Universal Robots PolyScope program: 28-pickAndPlace.urp

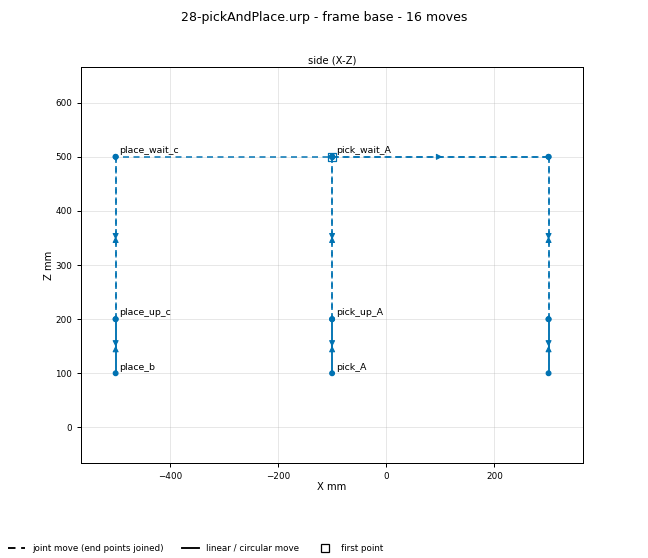
[picture p0: tool path of 28-pickAndPlace.urp in frame base, 16 of 16 moves have a stored position in this frame; points joined in program order, loops and branches not executed]
ProgramRoot directory=/home/ur/ursim-3.1/programs/basic training/28-pickAndPlace; kinematics=(a=[0, -0.425, -0.39225, 0, 0, 0], d=[0.08916, 0, 0, 0.10915, 0.09465, 0.0823], alpha=[1.5708, 0, 0, 1.5708, -1.5708, 0], deltaTheta=[0, 0, 0, 0, 0, 0], status=notInitialized); lastSavedInVersion=(project__name=Polyscope, major__version=3, minor__version=1, svn__revision=17195, build__date=Mar 11 2015, 13:02:28); name=28-pickAndPlace; programVersion=(project__name=Polyscope, major__version=3, minor__version=1, svn__revision=17195, build__date=Mar 11 2015, 13:02:28); robotEnvironmentFileName=default; serialNumberRobot=2014350001
  BeforeStart description=COMMAND_SEQUENCE_BEFORE_PROGRAM_START; name=BeforeStart
    Move cartesianAcceleration=1.2; cartesianSpeed=0.25; jointAcceleration=1.3962634015954636; jointSpeed=1.0471975511965976; sharedProcessMoveBlendRadius=0.025; motionType=JOINT_SPACE
      Waypoint blendRadius=0.05; cartesianAcceleration=1.2; cartesianSpeed=0.25; jointAcceleration=1.3962634015954636; jointSpeed=1.0471975511965976; nextMotionTime=2.0; stoppoint=true; useSharedBlendParameter=true; useSharedParameters=true; outputFlangePose=(pos=(x=-0.09999996819589972, y=-0.4000000526540407, z=0.5000000010103537), rot=(x=-0.0012210995530382433, y=3.1162764787073605, z=0.038892320957760594)); position=TCP in base x=-100 y=-400 z=500 mm, rx=-0.0012 ry=3.1163 rz=0.0389 rad; joints [-88.988, -79.302, -89.258, -102.845, 91.461, 0.95] deg; positionType=FIXED_POSITION; waypointPoseInFeatureCoordinates=(pos=(x=-0.0999999669318244, y=-0.4000001276702773, z=0.499999972698533), rot=(x=-0.0012210995530382489, y=3.1162764787073782, z=0.0388923209577583)); name=pick_wait_A
  MainProgram cartesianAcceleration=1.2; cartesianSpeed=0.25; jointAcceleration=1.3962634015954636; jointSpeed=1.0471975511965976; sharedProcessMoveBlendRadius=0.025; motionType=JOINT_SPACE
    If expr=ExpressionIONode; type=IF_NODE
      CallSubProgram subProgramNodeToCall=(SubProgramNode=(default=(keepHidden=false, keepSynchrnized=false, trackProgramExecution=false, name=sub_b)))
    If type=ELSE_NODE
      CallSubProgram subProgramNodeToCall=(SubProgramNode=(default=(keepHidden=false, keepSynchrnized=false, trackProgramExecution=false, name=sub_c)))
    CallSubProgram subProgramNodeToCall=(SubProgramNode=(default=(keepHidden=false, keepSynchrnized=false, trackProgramExecution=false, name=sub_a)))
  Event expression=ExpressionIONode
    Wait 
    Set 
  SubProgram name=sub_a
    Move cartesianAcceleration=1.2; cartesianSpeed=0.25; jointAcceleration=1.3962634015954636; jointSpeed=1.0471975511965976; sharedProcessMoveBlendRadius=0.025; motionType=JOINT_SPACE
      Waypoint blendRadius=0.05; cartesianAcceleration=1.2; cartesianSpeed=0.25; jointAcceleration=1.3962634015954636; jointSpeed=1.0471975511965976; nextMotionTime=2.0; stoppoint=true; useSharedBlendParameter=true; useSharedParameters=true; outputFlangePose=(pos=(x=-0.09999996819589972, y=-0.4000000526540407, z=0.5000000010103537), rot=(x=-0.0012210995530382433, y=3.1162764787073605, z=0.038892320957760594)); position=TCP in base x=-100 y=-400 z=500 mm, rx=-0.0012 ry=3.1163 rz=0.0389 rad; joints [-88.988, -79.302, -89.258, -102.845, 91.461, 0.95] deg; positionType=FIXED_POSITION; waypointPoseInFeatureCoordinates=(pos=(x=-0.0999999669318244, y=-0.4000001276702773, z=0.499999972698533), rot=(x=-0.0012210995530382489, y=3.1162764787073782, z=0.0388923209577583)); name=pick_wait_A
      Waypoint blendRadius=0.05; cartesianAcceleration=1.2; cartesianSpeed=0.25; jointAcceleration=1.3962634015954636; jointSpeed=1.0471975511965976; nextMotionTime=2.0; stoppoint=true; useSharedBlendParameter=true; useSharedParameters=true; outputFlangePose=(pos=(x=-0.09999996693182436, y=-0.40000012767028115, z=0.2000000005382103), rot=(x=-0.0012210995530365215, y=3.116276478707369, z=0.03889232095774556)); position=TCP in base x=-100 y=-400 z=200 mm, rx=-0.0012 ry=3.1163 rz=0.0389 rad; joints [-88.988, -88.3, -127.491, -55.614, 91.461, 0.95] deg; positionType=FIXED_POSITION; waypointPoseInFeatureCoordinates=(pos=(x=-0.09999996819589951, y=-0.40000005265404437, z=0.1999999632555712), rot=(x=-0.0012210995530369398, y=3.1162764787073427, z=0.0388923209577584)); name=pick_up_A
    Move cartesianAcceleration=1.2; cartesianSpeed=0.25; jointAcceleration=1.3962634015954636; jointSpeed=1.0471975511965976; sharedProcessMoveBlendRadius=0.025; motionType=CARTESIAN_SPACE
      Waypoint blendRadius=0.05; cartesianAcceleration=1.2; cartesianSpeed=0.25; jointAcceleration=1.3962634015954636; jointSpeed=1.0471975511965976; nextMotionTime=2.0; stoppoint=true; useSharedBlendParameter=true; useSharedParameters=true; outputFlangePose=(pos=(x=-0.0999999681958997, y=-0.4000000526540418, z=0.10000000081214921), rot=(x=-0.0012210995530447125, y=3.1162764787073605, z=0.038892320957759144)); position=TCP in base x=-100 y=-400 z=100 mm, rx=-0.0012 ry=3.1163 rz=0.0389 rad; joints [-88.988, -101.017, -134.096, -36.292, 91.461, 0.95] deg; positionType=FIXED_POSITION; waypointPoseInFeatureCoordinates=(pos=(x=-0.09999996708411972, y=-0.40000011440850547, z=0.10000011559988649), rot=(x=-0.0012211090279065008, y=3.1162764797380107, z=0.03889157798959221)); name=pick_A
      Waypoint blendRadius=0.05; cartesianAcceleration=1.2; cartesianSpeed=0.25; jointAcceleration=1.3962634015954636; jointSpeed=1.0471975511965976; nextMotionTime=2.0; stoppoint=true; useSharedBlendParameter=true; useSharedParameters=true; outputFlangePose=(pos=(x=-0.09999996693182436, y=-0.40000012767028115, z=0.2000000005382103), rot=(x=-0.0012210995530365215, y=3.116276478707369, z=0.03889232095774556)); position=TCP in base x=-100 y=-400 z=200 mm, rx=-0.0012 ry=3.1163 rz=0.0389 rad; joints [-88.988, -88.3, -127.491, -55.614, 91.461, 0.95] deg; positionType=FIXED_POSITION; waypointPoseInFeatureCoordinates=(pos=(x=-0.09999996819589951, y=-0.40000005265404437, z=0.1999999632555712), rot=(x=-0.0012210995530369398, y=3.1162764787073427, z=0.0388923209577584)); name=pick_up_A
    Move cartesianAcceleration=1.2; cartesianSpeed=0.25; jointAcceleration=1.3962634015954636; jointSpeed=1.0471975511965976; sharedProcessMoveBlendRadius=0.025; motionType=JOINT_SPACE
      Waypoint blendRadius=0.05; cartesianAcceleration=1.2; cartesianSpeed=0.25; jointAcceleration=1.3962634015954636; jointSpeed=1.0471975511965976; nextMotionTime=2.0; useSharedParameters=true; outputFlangePose=(pos=(x=-0.09999996819589972, y=-0.4000000526540407, z=0.5000000010103537), rot=(x=-0.0012210995530382433, y=3.1162764787073605, z=0.038892320957760594)); position=TCP in base x=-100 y=-400 z=500 mm, rx=-0.0012 ry=3.1163 rz=0.0389 rad; joints [-88.988, -79.302, -89.258, -102.845, 91.461, 0.95] deg; positionType=FIXED_POSITION; waypointPoseInFeatureCoordinates=(pos=(x=-0.0999999669318244, y=-0.4000001276702773, z=0.499999972698533), rot=(x=-0.0012210995530382489, y=3.1162764787073782, z=0.0388923209577583)); name=pick_wait_A
      Set 
  SubProgram name=sub_b
    Move cartesianAcceleration=1.2; cartesianSpeed=0.25; jointAcceleration=1.3962634015954636; jointSpeed=1.0471975511965976; sharedProcessMoveBlendRadius=0.025; motionType=JOINT_SPACE
      Waypoint blendRadius=0.05; cartesianAcceleration=1.2; cartesianSpeed=0.25; jointAcceleration=1.3962634015954636; jointSpeed=1.0471975511965976; nextMotionTime=2.0; useSharedParameters=true; outputFlangePose=(pos=(x=0.2999999995938011, y=-0.4000001276702728, z=0.49999997269853946), rot=(x=-0.0012210995530235833, y=3.11627647870737, z=0.03889232095775435)); position=TCP in base x=300 y=-400 z=500 mm, rx=-0.0012 ry=3.1163 rz=0.0389 rad; joints [-40.862, -90.996, -79.035, -99.819, 92.021, 49.096] deg; positionType=FIXED_POSITION; waypointPoseInFeatureCoordinates=(pos=(x=0.2999999592935196, y=-0.40000010776018363, z=0.4999999826709683), rot=(x=-0.001221022757481655, y=3.1162763421843853, z=0.03889217574522031)); name=place_wait_B
      Waypoint blendRadius=0.05; cartesianAcceleration=1.2; cartesianSpeed=0.25; jointAcceleration=1.3962634015954636; jointSpeed=1.0471975511965976; nextMotionTime=2.0; stoppoint=true; useSharedBlendParameter=true; useSharedParameters=true; outputFlangePose=(pos=(x=0.29999995929351975, y=-0.40000010776018347, z=0.20000000027822784), rot=(x=-0.0012210227574518974, y=3.1162763421844306, z=0.038892175745260965)); position=TCP in base x=300 y=-400 z=200 mm, rx=-0.0012 ry=3.1163 rz=0.0389 rad; joints [-40.862, -99.891, -115.262, -54.697, 92.021, 49.096] deg; positionType=FIXED_POSITION; waypointPoseInFeatureCoordinates=(pos=(x=0.2999999967409901, y=-0.40000014007290235, z=0.19999991255419813), rot=(x=-0.001221022757481655, y=3.1162763421843853, z=0.03889217574521508)); name=place_up_B
    Move cartesianAcceleration=1.2; cartesianSpeed=0.25; jointAcceleration=1.3962634015954636; jointSpeed=1.0471975511965976; sharedProcessMoveBlendRadius=0.025; motionType=CARTESIAN_SPACE
      Waypoint blendRadius=0.05; cartesianAcceleration=1.2; cartesianSpeed=0.25; jointAcceleration=1.3962634015954636; jointSpeed=1.0471975511965976; nextMotionTime=2.0; stoppoint=true; useSharedBlendParameter=true; useSharedParameters=true; outputFlangePose=(pos=(x=0.2999999967409869, y=-0.4000001400728996, z=0.1000000008121489), rot=(x=-0.0012210227574562102, y=3.1162763421844306, z=0.03889217574526195)); position=TCP in base x=300 y=-400 z=100 mm, rx=-0.0012 ry=3.1163 rz=0.0389 rad; joints [-40.862, -110.356, -120.826, -38.668, 92.021, 49.096] deg; positionType=FIXED_POSITION; waypointPoseInFeatureCoordinates=(pos=(x=0.3000000560345812, y=-0.4000001913379305, z=0.10000012111100774), rot=(x=-0.0012210357264685935, y=3.116275987797417, z=0.038891685033094876)); name=place_B
      Waypoint blendRadius=0.05; cartesianAcceleration=1.2; cartesianSpeed=0.25; jointAcceleration=1.3962634015954636; jointSpeed=1.0471975511965976; nextMotionTime=2.0; stoppoint=true; useSharedBlendParameter=true; useSharedParameters=true; outputFlangePose=(pos=(x=0.29999995929351975, y=-0.40000010776018347, z=0.20000000027822784), rot=(x=-0.0012210227574518974, y=3.1162763421844306, z=0.038892175745260965)); position=TCP in base x=300 y=-400 z=200 mm, rx=-0.0012 ry=3.1163 rz=0.0389 rad; joints [-40.862, -99.891, -115.262, -54.697, 92.021, 49.096] deg; positionType=FIXED_POSITION; waypointPoseInFeatureCoordinates=(pos=(x=0.2999999967409901, y=-0.40000014007290235, z=0.19999991255419813), rot=(x=-0.001221022757481655, y=3.1162763421843853, z=0.03889217574521508)); name=place_up_B
    Move cartesianAcceleration=1.2; cartesianSpeed=0.25; jointAcceleration=1.3962634015954636; jointSpeed=1.0471975511965976; sharedProcessMoveBlendRadius=0.025; motionType=JOINT_SPACE
      Waypoint blendRadius=0.05; cartesianAcceleration=1.2; cartesianSpeed=0.25; jointAcceleration=1.3962634015954636; jointSpeed=1.0471975511965976; nextMotionTime=2.0; useSharedParameters=true; outputFlangePose=(pos=(x=0.2999999995938011, y=-0.4000001276702728, z=0.49999997269853946), rot=(x=-0.0012210995530235833, y=3.11627647870737, z=0.03889232095775435)); position=TCP in base x=300 y=-400 z=500 mm, rx=-0.0012 ry=3.1163 rz=0.0389 rad; joints [-40.862, -90.996, -79.035, -99.819, 92.021, 49.096] deg; positionType=FIXED_POSITION; waypointPoseInFeatureCoordinates=(pos=(x=0.2999999592935196, y=-0.40000010776018363, z=0.4999999826709683), rot=(x=-0.001221022757481655, y=3.1162763421843853, z=0.03889217574522031)); name=place_wait_B
  SubProgram name=sub_c
    Move cartesianAcceleration=1.2; cartesianSpeed=0.25; jointAcceleration=1.3962634015954636; jointSpeed=1.0471975511965976; sharedProcessMoveBlendRadius=0.025; motionType=JOINT_SPACE
      Waypoint blendRadius=0.05; cartesianAcceleration=1.2; cartesianSpeed=0.25; jointAcceleration=1.3962634015954636; jointSpeed=1.0471975511965976; nextMotionTime=2.0; useSharedParameters=true; outputFlangePose=(pos=(x=-0.4999999998054968, y=-0.40000010776019246, z=0.4999999826709834), rot=(x=-0.001221022757489431, y=3.1162763421844115, z=0.03889217574523564)); position=TCP in base x=-500 y=-400 z=500 mm, rx=-0.0012 ry=3.1163 rz=0.0389 rad; joints [-131.542, -112.233, -52.539, -107.251, 90.126, -41.589] deg; positionType=FIXED_POSITION; waypointPoseInFeatureCoordinates=(pos=(x=-0.5000000953689041, y=-0.40000011657723855, z=0.4999999157130972), rot=(x=-0.0012208175643654505, y=3.116276278412111, z=0.03889241911004195)); name=place_wait_c
      Waypoint blendRadius=0.05; cartesianAcceleration=1.2; cartesianSpeed=0.25; jointAcceleration=1.3962634015954636; jointSpeed=1.0471975511965976; nextMotionTime=2.0; stoppoint=true; useSharedBlendParameter=true; useSharedParameters=true; outputFlangePose=(pos=(x=-0.5000000953689022, y=-0.4000001165772364, z=0.20000000050812997), rot=(x=-0.0012208175644618617, y=3.1162762784121854, z=0.038892419110114325)); position=TCP in base x=-500 y=-400 z=200 mm, rx=-0.0012 ry=3.1163 rz=0.0389 rad; joints [-131.542, -116.881, -90.871, -64.271, 90.126, -41.589] deg; positionType=FIXED_POSITION; waypointPoseInFeatureCoordinates=(pos=(x=-0.5000000607401942, y=-0.40000007758696715, z=0.20000003652729953), rot=(x=-0.0012208175643609084, y=3.11627627841208, z=0.03889241911005109)); name=place_up_c
    Move cartesianAcceleration=1.2; cartesianSpeed=0.25; jointAcceleration=1.3962634015954636; jointSpeed=1.0471975511965976; sharedProcessMoveBlendRadius=0.025; motionType=CARTESIAN_SPACE
      Waypoint blendRadius=0.05; cartesianAcceleration=1.2; cartesianSpeed=0.25; jointAcceleration=1.3962634015954636; jointSpeed=1.0471975511965976; nextMotionTime=2.0; stoppoint=true; useSharedBlendParameter=true; useSharedParameters=true; outputFlangePose=(pos=(x=-0.5000000607401927, y=-0.4000000775869654, z=0.10000000101628408), rot=(x=-0.0012208175644851543, y=3.1162762784121942, z=0.03889241911011709)); position=TCP in base x=-500 y=-400 z=100 mm, rx=-0.0012 ry=3.1163 rz=0.0389 rad; joints [-131.542, -124.449, -95.914, -51.659, 90.126, -41.589] deg; positionType=FIXED_POSITION; waypointPoseInFeatureCoordinates=(pos=(x=-0.5000000521643437, y=-0.4000000679389194, z=0.10000011853029817), rot=(x=-0.0012208175643656706, y=3.1162762784120708, z=0.03889241911006023)); name=place_b
      Waypoint blendRadius=0.05; cartesianAcceleration=1.2; cartesianSpeed=0.25; jointAcceleration=1.3962634015954636; jointSpeed=1.0471975511965976; nextMotionTime=2.0; stoppoint=true; useSharedBlendParameter=true; useSharedParameters=true; outputFlangePose=(pos=(x=-0.5000000953689022, y=-0.4000001165772364, z=0.20000000050812997), rot=(x=-0.0012208175644618617, y=3.1162762784121854, z=0.038892419110114325)); position=TCP in base x=-500 y=-400 z=200 mm, rx=-0.0012 ry=3.1163 rz=0.0389 rad; joints [-131.542, -116.881, -90.871, -64.271, 90.126, -41.589] deg; positionType=FIXED_POSITION; waypointPoseInFeatureCoordinates=(pos=(x=-0.5000000607401942, y=-0.40000007758696715, z=0.20000003652729953), rot=(x=-0.0012208175643609084, y=3.11627627841208, z=0.03889241911005109)); name=place_up_c
    Move cartesianAcceleration=1.2; cartesianSpeed=0.25; jointAcceleration=1.3962634015954636; jointSpeed=1.0471975511965976; sharedProcessMoveBlendRadius=0.025; motionType=JOINT_SPACE
      Waypoint blendRadius=0.05; cartesianAcceleration=1.2; cartesianSpeed=0.25; jointAcceleration=1.3962634015954636; jointSpeed=1.0471975511965976; nextMotionTime=2.0; useSharedParameters=true; outputFlangePose=(pos=(x=-0.4999999998054968, y=-0.40000010776019246, z=0.4999999826709834), rot=(x=-0.001221022757489431, y=3.1162763421844115, z=0.03889217574523564)); position=TCP in base x=-500 y=-400 z=500 mm, rx=-0.0012 ry=3.1163 rz=0.0389 rad; joints [-131.542, -112.233, -52.539, -107.251, 90.126, -41.589] deg; positionType=FIXED_POSITION; waypointPoseInFeatureCoordinates=(pos=(x=-0.5000000953689041, y=-0.40000011657723855, z=0.4999999157130972), rot=(x=-0.0012208175643654505, y=3.116276278412111, z=0.03889241911004195)); name=place_wait_c
